FUNCTION_BLOCK CRANE_SELECTOR (* Service Interface Function Block Type *)
  (* Standard: 61499-2 *)
  (* Version 1.0, 2019-04-04, adeel *)
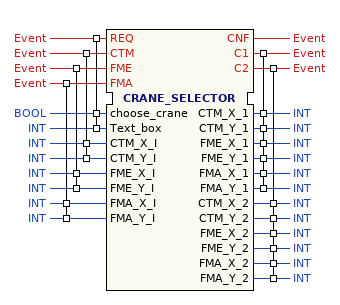
  EVENT_INPUT
    REQ WITH choose_crane, Text_box; (* Service Request *)
    CTM WITH CTM_X_I, CTM_Y_I;
    FME WITH FME_X_I, FME_Y_I;
    FMA WITH FMA_X_I, FMA_Y_I;
  END_EVENT
  EVENT_OUTPUT
    CNF; (* Confirmation of Requested Service *)
    C1 WITH CTM_X_1, CTM_Y_1, FME_X_1, FME_Y_1, FMA_X_1, FMA_Y_1;
    C2 WITH CTM_X_2, CTM_Y_2, FME_X_2, FME_Y_2, FMA_X_2, FMA_Y_2;
  END_EVENT
  VAR_INPUT
    choose_crane : BOOL;
    Text_box : INT;
    CTM_X_I : INT;
    CTM_Y_I : INT;
    FME_X_I : INT;
    FME_Y_I : INT;
    FMA_X_I : INT;
    FMA_Y_I : INT;
  END_VAR
  VAR_OUTPUT
    CTM_X_1 : INT;
    CTM_Y_1 : INT;
    FME_X_1 : INT;
    FME_Y_1 : INT;
    FMA_X_1 : INT;
    FMA_Y_1 : INT;
    CTM_X_2 : INT;
    CTM_Y_2 : INT;
    FME_X_2 : INT;
    FME_Y_2 : INT;
    FMA_X_2 : INT;
    FMA_Y_2 : INT;
  END_VAR
  SERVICE APPLICATION/RESOURCE (* Service Interface Function Block Type *)
    SEQUENCE normal_establishment
      APPLICATION.INIT+(PARAMS) -> RESOURCE.initialize(PARAMS) -> APPLICATION.INITO+();
    END_SEQUENCE
    SEQUENCE unsuccessful_establishment
      APPLICATION.INIT+(PARAMS) -> RESOURCE.initialize(PARAMS) -> APPLICATION.INITO-(STATUS);
    END_SEQUENCE
    SEQUENCE request_confirm
      APPLICATION.REQ+(SD) -> RESOURCE.request(SD) -> APPLICATION.CNF+(RD);
    END_SEQUENCE
    SEQUENCE request_inhibited
      APPLICATION.REQ-(SD) -> APPLICATION.CNF-(STATUS);
    END_SEQUENCE
    SEQUENCE request_error
      APPLICATION.REQ+(SD) -> RESOURCE.request(SD) -> APPLICATION.CNF-(STATUS);
    END_SEQUENCE
    SEQUENCE indication_response
      RESOURCE.indicate(RD) -> APPLICATION.IND+(RD);
      APPLICATION.RSP(QI,SD) -> RESOURCE.response(QI,SD);
    END_SEQUENCE
    SEQUENCE indication_inhibited
      RESOURCE.indicate(RD,QI=FALSE) -> RESOURCE.inhibited();
    END_SEQUENCE
    SEQUENCE error_indication
      RESOURCE.error(STATUS) -> APPLICATION.IND-(STATUS);
    END_SEQUENCE
    SEQUENCE application_initiated_termination
      APPLICATION.INIT-() -> RESOURCE.terminate() -> APPLICATION.INITO-(STATUS);
    END_SEQUENCE
    SEQUENCE resource_initiated_termination
      -> APPLICATION.INITO-(STATUS);
    END_SEQUENCE
  END_SERVICE
END_FUNCTION_BLOCK
